TYPE ST_Event :
STRUCT
	eEventType : E_EventType;
	eEventSeverity : TcEventseverity;
	nEventIdentity : UDINT;
	sEventText : STRING(255);
	dtTimeStamp : DATE_AND_TIME;
END_STRUCT
END_TYPE

(* stored: Version 1.1.0.1, ProductVersion 3.1.4024.16
   DUT ST_Event: Id {bd760163-ad47-46a0-b3ca-63c139b9acfd} *)
